{attribute addProperty BoxType "EM3701-0000-0016"}
{attribute addProperty Id "StatusAT %I*Status_3D195A321621ValueAT %I*INT16217"}
{attribute addProperty CRC "3613813698"}
{attribute addProperty SizeInBites "32"}
{attribute addProperty SizeInBytes "4"}
TYPE AI_Inputs_D7666BC2 :
STRUCT
	{attribute addProperty Name "Status"}
	Status AT %I* : Status_3D195A32;
	{attribute addProperty Name "Value"}
	Value AT %I* : INT;
END_STRUCT
END_TYPE

(* stored: Version 1.2.0.0, ProductVersion 3.1.4024.9
   DUT AI_Inputs_D7666BC2: Id {2a6defc0-c2b4-43af-9117-7adbb9997635} *)
